Staubli VAL3: object.pjx

--- object.pjx ---
Parameters version=s7.6 stackSize=5000 millimeterUnit=true
Program file=start.pgx
Program file=stop.pgx
Data file=object.dtx

--- start.pgx ---
program start()
begin

end

--- stop.pgx ---
program stop()
begin

end
